// TIA Portal V21 export
DATA_BLOCK "IEC_Counter_0_DB_3"   // DB153
{ S7_Optimized_Access := 'TRUE' }
// stored: InstanceOfName IEC_COUNTER, OfSystemLibElement IEC_COUNTER, OfSystemLibVersion 1.0
"IEC_COUNTER"
   // VAR RETAIN
   //    CU : Bool;
   //    CD : Bool;
   //    R : Bool;
   //    LD : Bool;
   //    QU : Bool;
   //    QD : Bool;
   //    PV : Int;
   //    CV : Int;
   // END_VAR
BEGIN
END_DATA_BLOCK
